FUNCTION_BLOCK EA_2_rightSwitch
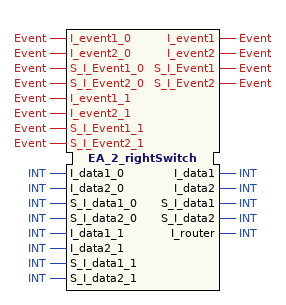
  EVENT_INPUT
    I_event1_0;
    I_event2_0;
    S_I_Event1_0;
    S_I_Event2_0;
    I_event1_1;
    I_event2_1;
    S_I_Event1_1;
    S_I_Event2_1;
  END_EVENT
  EVENT_OUTPUT
    I_event1;
    I_event2;
    S_I_Event1;
    S_I_Event2;
  END_EVENT
  VAR_INPUT
    I_data1_0 : INT;
    I_data2_0 : INT;
    S_I_data1_0 : INT;
    S_I_data2_0 : INT;
    I_data1_1 : INT;
    I_data2_1 : INT;
    S_I_data1_1 : INT;
    S_I_data2_1 : INT;
  END_VAR
  VAR_OUTPUT
    I_data1 : INT;
    I_data2 : INT;
    S_I_data1 : INT;
    S_I_data2 : INT;
    I_router : INT;
  END_VAR
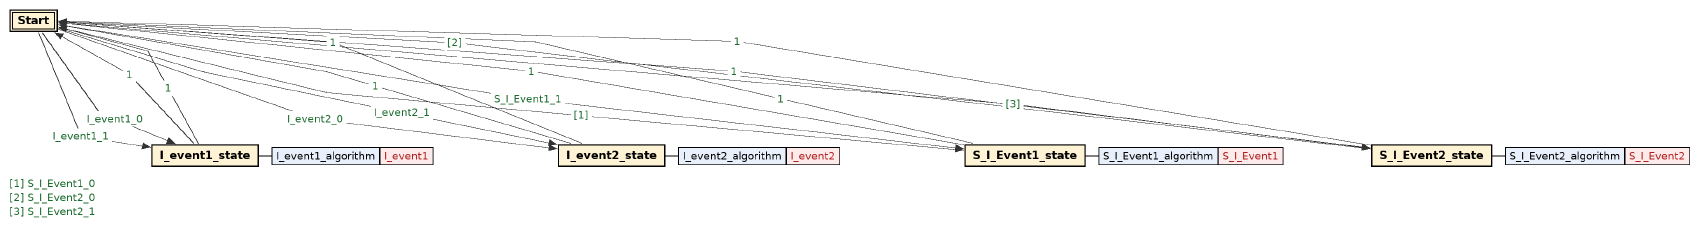
  EC_STATES
    Start;
    I_event1_state : I_event1_algorithm -> I_event1;
    I_event2_state : I_event2_algorithm -> I_event2;
    S_I_Event1_state : S_I_Event1_algorithm -> S_I_Event1;
    S_I_Event2_state : S_I_Event2_algorithm -> S_I_Event2;
    I_event1_state : I_event1_algorithm -> I_event1;
    I_event2_state : I_event2_algorithm -> I_event2;
    S_I_Event1_state : S_I_Event1_algorithm -> S_I_Event1;
    S_I_Event2_state : S_I_Event2_algorithm -> S_I_Event2;
  END_STATES
  EC_TRANSITIONS
    I_event1_state TO Start := 1;
    Start TO I_event1_state := I_event1_0;
    I_event2_state TO Start := 1;
    Start TO I_event2_state := I_event2_0;
    S_I_Event1_state TO Start := 1;
    Start TO S_I_Event1_state := S_I_Event1_0;
    S_I_Event2_state TO Start := 1;
    Start TO S_I_Event2_state := S_I_Event2_0;
    I_event1_state TO Start := 1;
    Start TO I_event1_state := I_event1_1;
    I_event2_state TO Start := 1;
    Start TO I_event2_state := I_event2_1;
    S_I_Event1_state TO Start := 1;
    Start TO S_I_Event1_state := S_I_Event1_1;
    S_I_Event2_state TO Start := 1;
    Start TO S_I_Event2_state := S_I_Event2_1;
  END_TRANSITIONS
  ALGORITHM I_event1_algorithm IN ST:
I_data1 := I_data1_0;&#38;#10;I_data2 := I_data2_0;&#38;#10;S_I_data1 := S_I_data1_0;&#38;#10;S_I_data2 := S_I_data2_0;&#38;#10;I_router := 0;&#38;#10;
  END_ALGORITHM
  ALGORITHM I_event2_algorithm IN ST:
I_data1 := I_data1_0;&#38;#10;I_data2 := I_data2_0;&#38;#10;S_I_data1 := S_I_data1_0;&#38;#10;S_I_data2 := S_I_data2_0;&#38;#10;I_router := 0;&#38;#10;
  END_ALGORITHM
  ALGORITHM S_I_Event1_algorithm IN ST:
I_data1 := I_data1_0;&#38;#10;I_data2 := I_data2_0;&#38;#10;S_I_data1 := S_I_data1_0;&#38;#10;S_I_data2 := S_I_data2_0;&#38;#10;I_router := 0;&#38;#10;
  END_ALGORITHM
  ALGORITHM S_I_Event2_algorithm IN ST:
I_data1 := I_data1_0;&#38;#10;I_data2 := I_data2_0;&#38;#10;S_I_data1 := S_I_data1_0;&#38;#10;S_I_data2 := S_I_data2_0;&#38;#10;I_router := 0;&#38;#10;
  END_ALGORITHM
  ALGORITHM I_event1_algorithm IN ST:
I_data1 := I_data1_1;&#38;#10;I_data2 := I_data2_1;&#38;#10;S_I_data1 := S_I_data1_1;&#38;#10;S_I_data2 := S_I_data2_1;&#38;#10;I_router := 1;&#38;#10;
  END_ALGORITHM
  ALGORITHM I_event2_algorithm IN ST:
I_data1 := I_data1_1;&#38;#10;I_data2 := I_data2_1;&#38;#10;S_I_data1 := S_I_data1_1;&#38;#10;S_I_data2 := S_I_data2_1;&#38;#10;I_router := 1;&#38;#10;
  END_ALGORITHM
  ALGORITHM S_I_Event1_algorithm IN ST:
I_data1 := I_data1_1;&#38;#10;I_data2 := I_data2_1;&#38;#10;S_I_data1 := S_I_data1_1;&#38;#10;S_I_data2 := S_I_data2_1;&#38;#10;I_router := 1;&#38;#10;
  END_ALGORITHM
  ALGORITHM S_I_Event2_algorithm IN ST:
I_data1 := I_data1_1;&#38;#10;I_data2 := I_data2_1;&#38;#10;S_I_data1 := S_I_data1_1;&#38;#10;S_I_data2 := S_I_data2_1;&#38;#10;I_router := 1;&#38;#10;
  END_ALGORITHM
END_FUNCTION_BLOCK
